FUNCTION_BLOCK Equipamento_On_Off (* Composite Function Block Type *)
  (* Standard: 61499-2 *)
  (* Version 0.0, 1/26/2026, Schneider Electric, template *)
  PACKAGE Hidryco.HidrycoLib;
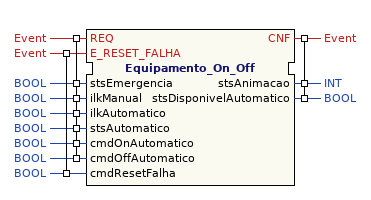
  EVENT_INPUT
    REQ WITH ilkManual, ilkAutomatico, cmdOnAutomatico, cmdOffAutomatico, stsAutomatico, stsEmergencia; (* Normal Execution Request *)
    E_RESET_FALHA WITH cmdResetFalha;
  END_EVENT
  EVENT_OUTPUT
    CNF WITH stsAnimacao, stsDisponivelAutomatico;
  END_EVENT
  VAR_INPUT
    stsEmergencia : BOOL;
    ilkManual : BOOL;
    ilkAutomatico : BOOL;
    stsAutomatico : BOOL;
    cmdOnAutomatico : BOOL;
    cmdOffAutomatico : BOOL;
    cmdResetFalha : BOOL;
  END_VAR
  VAR_OUTPUT
    stsAnimacao : INT;
    stsDisponivelAutomatico : BOOL;
  END_VAR
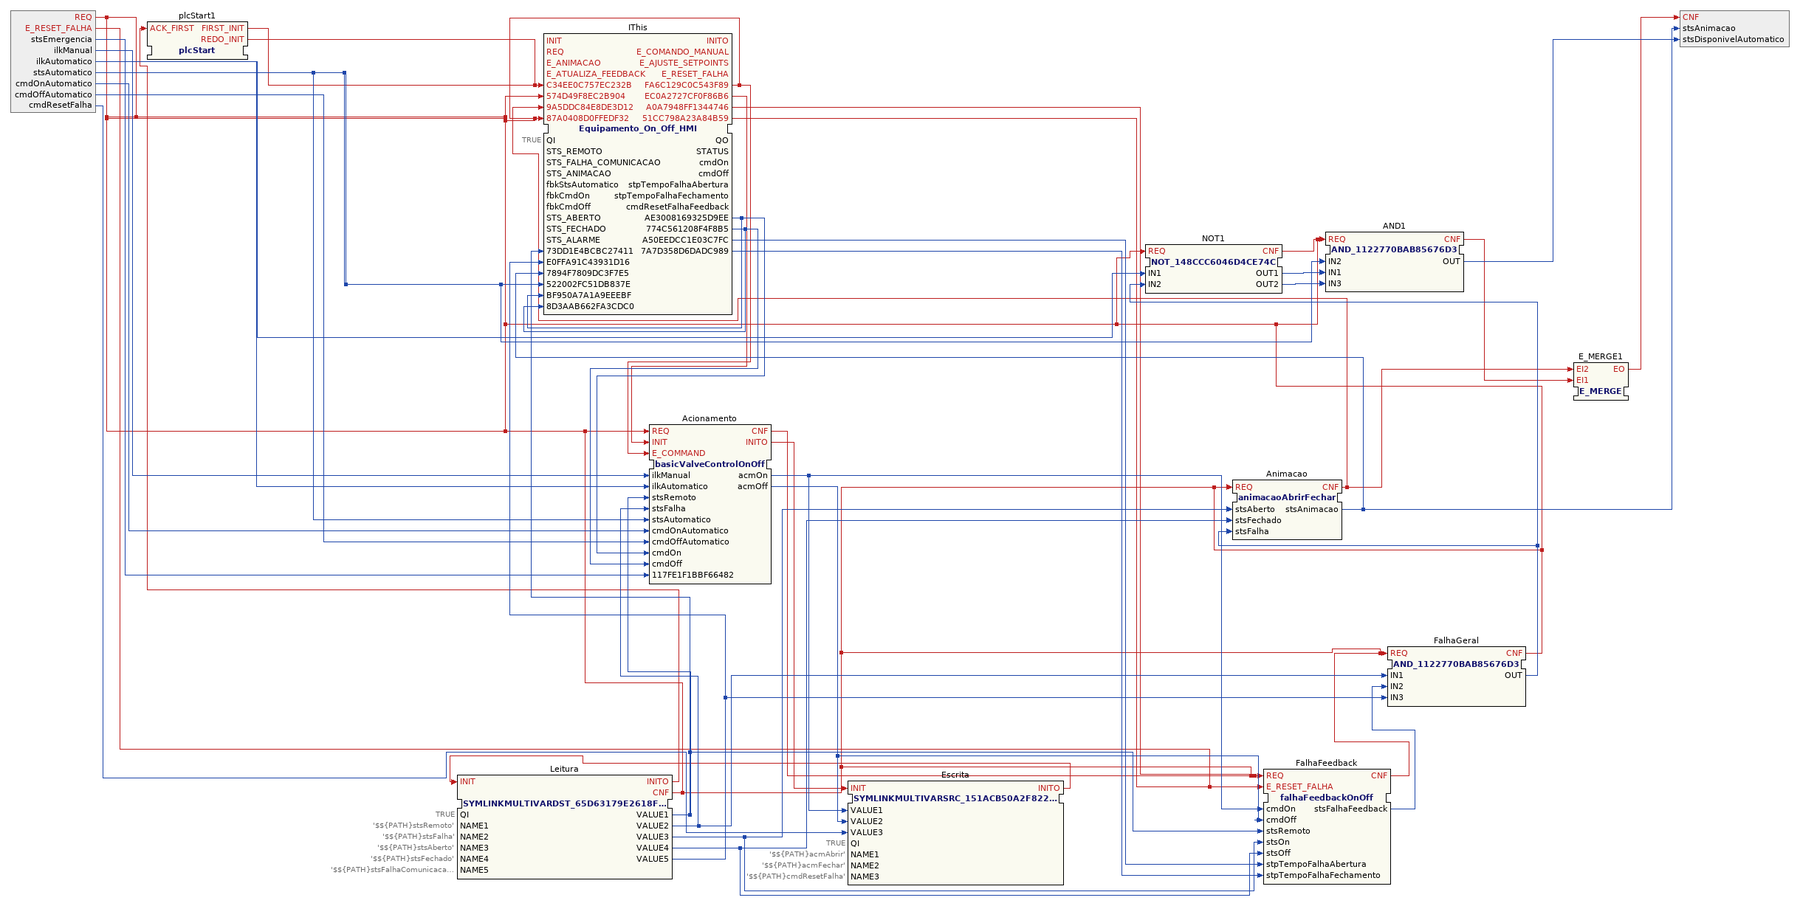
  FBS
    Acionamento : basicValveControlOnOff;
    IThis : Equipamento_On_Off_HMI(QI := TRUE);
    Animacao : animacaoAbrirFechar;
    FalhaFeedback : falhaFeedbackOnOff;
    FalhaGeral : AND_1122770BAB85676D3; {SET_ATTRIBUTE(Configuration.GenericFBType.InterfaceParams, Runtime.Standard#CNT:=3)}
    Leitura : SYMLINKMULTIVARDST_65D63179E2618F5E(QI := TRUE, NAME1 := '$${PATH}stsRemoto', NAME2 := '$${PATH}stsFalha', NAME3 := '$${PATH}stsAberto', NAME4 := '$${PATH}stsFechado', NAME5 := '$${PATH}stsFalhaComunicacao'); {SET_ATTRIBUTE(Configuration.GenericFBType.InterfaceParams, Runtime.System#I:=5;VALUE${I$}:BOOL,BOOL,BOOL,BOOL,BOOL)}
    plcStart1 : plcStart;
    Escrita : SYMLINKMULTIVARSRC_151ACB50A2F8223B2(QI := TRUE, NAME1 := '$${PATH}acmAbrir', NAME2 := '$${PATH}acmFechar', NAME3 := '$${PATH}cmdResetFalha'); {SET_ATTRIBUTE(Configuration.GenericFBType.InterfaceParams, Runtime.System#I:=3;VALUE${I$}:BOOL,BOOL,BOOL)}
    AND1 : AND_1122770BAB85676D3; {SET_ATTRIBUTE(Configuration.GenericFBType.InterfaceParams, Runtime.Standard#CNT:=3)}
    NOT1 : NOT_148CCC6046D4CE74C; {SET_ATTRIBUTE(Configuration.GenericFBType.InterfaceParams, Runtime.Standard#CNT:=2)}
    E_MERGE1 : E_MERGE;
  END_FBS
  EVENT_CONNECTIONS
    REQ TO Acionamento.REQ;
    Acionamento.CNF TO FalhaFeedback.REQ;
    E_RESET_FALHA TO FalhaFeedback.E_RESET_FALHA;
    Leitura.INITO TO plcStart1.ACK_FIRST;
    Leitura.CNF TO FalhaFeedback.REQ;
    Leitura.CNF TO Animacao.REQ;
    Animacao.CNF TO E_MERGE1.EI2;
    plcStart1.FIRST_INIT TO IThis.C34EE0C757EC232B;
    plcStart1.REDO_INIT TO IThis.C34EE0C757EC232B;
    Leitura.CNF TO IThis.574D49F8EC2B904;
    Animacao.CNF TO IThis.9A5DDC84E8DE3D12;
    IThis.FA6C129C0C543F89 TO IThis.87A0408D0FFEDF32;
    REQ TO IThis.87A0408D0FFEDF32;
    IThis.EC0A2727CF0F86B6 TO Acionamento.INIT;
    IThis.FA6C129C0C543F89 TO Acionamento.E_COMMAND;
    IThis.A0A7948FF1344746 TO FalhaFeedback.REQ;
    IThis.51CC798A23A84B59 TO FalhaFeedback.E_RESET_FALHA;
    E_MERGE1.EO TO CNF;
    REQ TO AND1.REQ;
    AND1.CNF TO E_MERGE1.EI1;
    REQ TO NOT1.REQ;
    NOT1.CNF TO AND1.REQ;
    FalhaFeedback.CNF TO FalhaGeral.REQ;
    Leitura.CNF TO FalhaGeral.REQ;
    FalhaGeral.CNF TO Animacao.REQ;
    FalhaGeral.CNF TO NOT1.REQ;
    Acionamento.INITO TO Escrita.INIT;
    Escrita.INITO TO Leitura.INIT;
  END_CONNECTIONS
  DATA_CONNECTIONS
    ilkManual TO Acionamento.ilkManual;
    ilkAutomatico TO Acionamento.ilkAutomatico;
    Acionamento.acmOn TO FalhaFeedback.cmdOn;
    Acionamento.acmOff TO FalhaFeedback.cmdOff;
    Leitura.VALUE1 TO Acionamento.stsRemoto;
    Leitura.VALUE1 TO FalhaFeedback.stsRemoto;
    Leitura.VALUE2 TO Acionamento.stsFalha;
    Leitura.VALUE3 TO Animacao.stsAberto;
    Leitura.VALUE3 TO FalhaFeedback.stsOn;
    Leitura.VALUE4 TO Animacao.stsFechado;
    Leitura.VALUE4 TO FalhaFeedback.stsOff;
    Animacao.stsAnimacao TO stsAnimacao;
    stsAutomatico TO Acionamento.stsAutomatico;
    cmdOnAutomatico TO Acionamento.cmdOnAutomatico;
    cmdOffAutomatico TO Acionamento.cmdOffAutomatico;
    Leitura.VALUE1 TO IThis.73DD1E4BCBC27411;
    Leitura.VALUE5 TO IThis.E0FFA91C43931D16;
    Animacao.stsAnimacao TO IThis.7894F7809DC3F7E5;
    stsAutomatico TO IThis.522002FC51DB837E;
    IThis.AE3008169325D9EE TO IThis.BF950A7A1A9EEEBF;
    IThis.774C561208F4F8B5 TO IThis.8D3AAB662FA3CDC0;
    IThis.AE3008169325D9EE TO Acionamento.cmdOn;
    IThis.774C561208F4F8B5 TO Acionamento.cmdOff;
    IThis.A50EEDCC1E03C7FC TO FalhaFeedback.stpTempoFalhaAbertura;
    IThis.7A7D358D6DADC989 TO FalhaFeedback.stpTempoFalhaFechamento;
    stsAutomatico TO AND1.IN2;
    AND1.OUT TO stsDisponivelAutomatico;
    ilkAutomatico TO NOT1.IN1;
    NOT1.OUT1 TO AND1.IN1;
    NOT1.OUT2 TO AND1.IN3;
    Leitura.VALUE2 TO FalhaGeral.IN1;
    FalhaFeedback.stsFalhaFeedback TO FalhaGeral.IN2;
    FalhaGeral.OUT TO Animacao.stsFalha;
    FalhaGeral.OUT TO NOT1.IN2;
    Leitura.VALUE5 TO FalhaGeral.IN3;
    Acionamento.acmOn TO Escrita.VALUE1;
    Acionamento.acmOff TO Escrita.VALUE2;
    cmdResetFalha TO Escrita.VALUE3;
    stsEmergencia TO Acionamento.117FE1F1BBF66482;
  END_CONNECTIONS
END_FUNCTION_BLOCK
